// TIA Portal V20 export
TYPE "typeCmControlNode"
// stored: Namespace Unit1.Em10
   STRUCT
      interlock : "Unit1.Em10.typeCmControlNodeInterlock";
   END_STRUCT;
END_TYPE
